(* Schneider Machine Expert - Basic project Motor_StartStop_Overload_TM221CE16T, file version 3.0.0.0 *)
(* ProjectInformations: Name=New project *)

HARDWARE
  Cpu 0: TM221CE16T
  EthernetConfiguration: NetworkName=M221, IpAllocationMode=FixedAddress, IpAddress=0.0.0.0, SubnetMask=0.0.0.0
  SerialLineConfiguration: Baud=Baud19200, Parity=ParityEven, DataBits=DataBits8, StopBits=StopBits1, PhysicalMedium=PhysicalMediumRs485, TransmissionMode=TransmissionModeModbusRtu, SlaveId=1, Addressing=SlaveAddressing
  MastTask: UsePeriodScanMode=false, PeriodScan=100
  FastTask: Period=255
  CpuBehavior: StartingMode=StartAsPreviousState, AutoSaveRamOnEeprom=true, WatchdogPeriod=250

SYMBOLS  (address, symbol, comment, settings)
  %M0       SYSTEM_READY
  %M1       MOTOR_RUNNING
  %M2       OVERLOAD_ALARM
  %M3       ANY_ALARM
  %S0       SB_COLDSTART  "Indicates or executes a cold start (data initialized to default values)"
  %S1       SB_WARMSTART  "Indicates there was a warm start with data backup"
  %TM0        [Preset=3, Base=OneSecond]
  %TM1        [Preset=5, Base=HundredMilliseconds]
  %I0.0     EMERGENCY_PB

POU Motor Control
  (* SectionNumber=0 *)

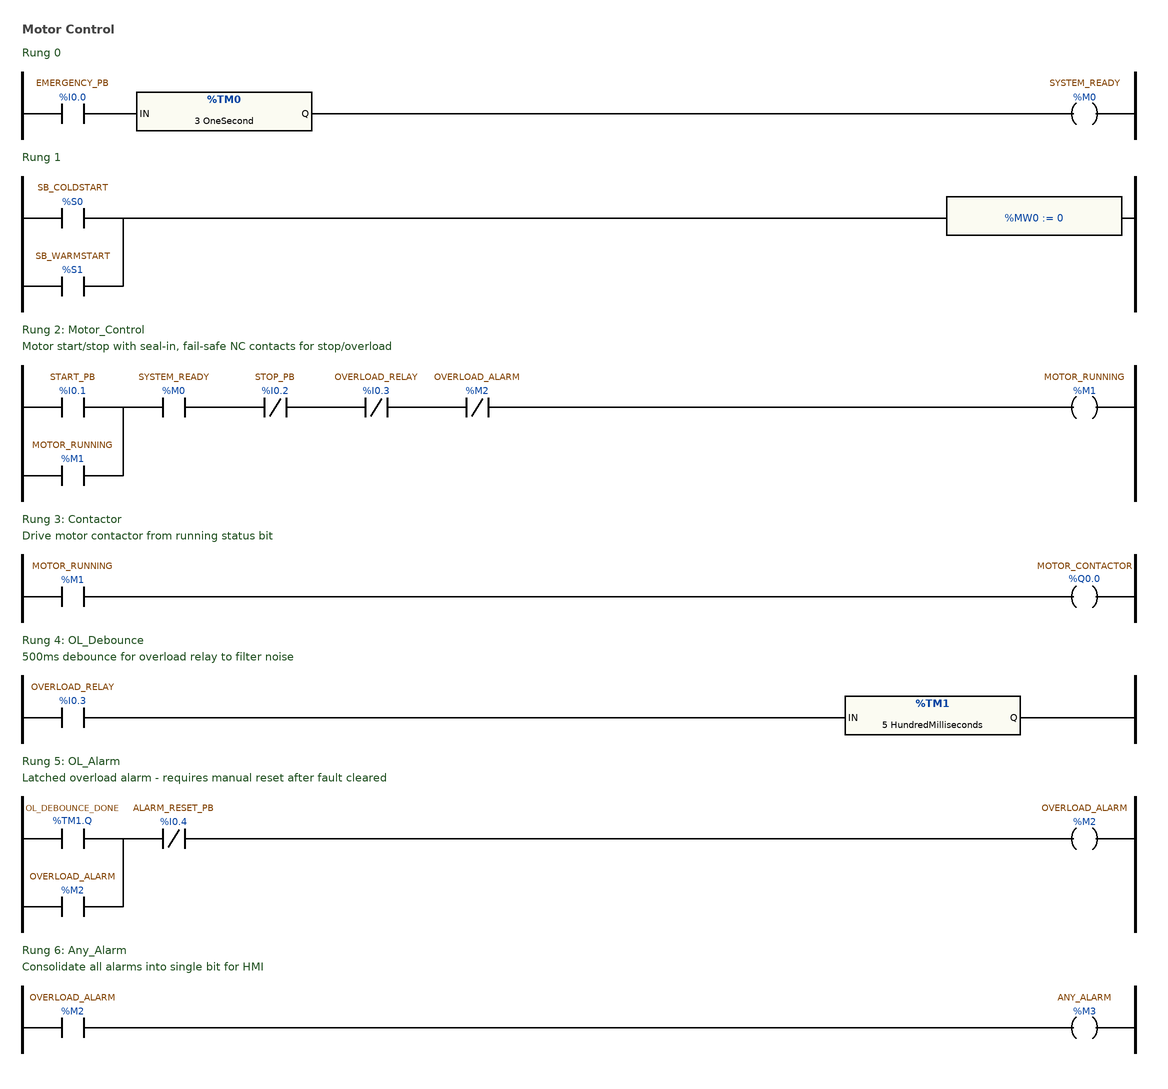

// Rung 0
  BLK %TM0
  LD %I0.0                (* EMERGENCY_PB *)
  IN
  OUT_BLK
  LD Q
  ST %M0                  (* SYSTEM_READY *)
  END_BLK
  // as ST:
  //   %TM0(IN := EMERGENCY_PB);
  //   SYSTEM_READY := %TM0.Q;

// Rung 1
  LD %S0                  (* SB_COLDSTART *)
  OR %S1                  (* SB_WARMSTART *)
  [ %MW0 := 0 ]
  // as ST:
  //   IF SB_COLDSTART OR SB_WARMSTART THEN %MW0 := 0; END_IF;

// Rung 2: Motor_Control
// Motor start/stop with seal-in, fail-safe NC contacts for stop/overload
  LD %I0.1                (* Start Pushbutton *)
  OR %M1                  (* MOTOR_RUNNING - Seal-in *)
  AND %M0                 (* SYSTEM_READY - System Ready *)
  ANDN %I0.2              (* Stop Button NC *)
  ANDN %I0.3              (* Overload OK *)
  ANDN %M2                (* OVERLOAD_ALARM - No Alarm *)
  ST %M1                  (* MOTOR_RUNNING - Motor Running *)
  // %I0.1: Start Pushbutton
  // %M0: System Ready
  // %I0.2: Stop Button NC
  // %I0.3: Overload OK
  // %M2: No Alarm
  // %M1: Motor Running
  // %M1: Seal-in
  // as ST:
  //   MOTOR_RUNNING := (%I0.1 OR MOTOR_RUNNING) AND SYSTEM_READY AND NOT %I0.2 AND NOT %I0.3 AND NOT OVERLOAD_ALARM;

// Rung 3: Contactor
// Drive motor contactor from running status bit
  LD %M1                  (* MOTOR_RUNNING - Motor Running *)
  ST %Q0.0                (* Motor Contactor *)
  // %M1: Motor Running
  // %Q0.0: Motor Contactor
  // as ST:
  //   %Q0.0 := MOTOR_RUNNING;

// Rung 4: OL_Debounce
// 500ms debounce for overload relay to filter noise
  BLK %TM1                (* Overload Debounce Timer *)
  LD %I0.3                (* Overload Relay Tripped *)
  IN
  OUT_BLK
  END_BLK
  // %I0.3: Overload Tripped
  // %TM1: 500ms Debounce
  // as ST:
  //   %TM1(IN := %I0.3);

// Rung 5: OL_Alarm
// Latched overload alarm - requires manual reset after fault cleared
  LD %TM1.Q               (* Debounce Timer Done *)
  OR %M2                  (* OVERLOAD_ALARM - Seal-in Alarm *)
  ANDN %I0.4              (* Reset Not Pressed *)
  ST %M2                  (* OVERLOAD_ALARM - Overload Alarm *)
  // %TM1.Q: Debounce Done
  // %I0.4: Reset Not Pressed
  // %M2: Overload Alarm
  // %M2: Seal-in
  // as ST:
  //   OVERLOAD_ALARM := (%TM1.Q OR OVERLOAD_ALARM) AND NOT %I0.4;

// Rung 6: Any_Alarm
// Consolidate all alarms into single bit for HMI
  LD %M2                  (* OVERLOAD_ALARM - Overload Alarm *)
  ST %M3                  (* ANY_ALARM - Any Alarm *)
  // %M2: Overload Alarm
  // %M3: Any Alarm
  // as ST:
  //   ANY_ALARM := OVERLOAD_ALARM;

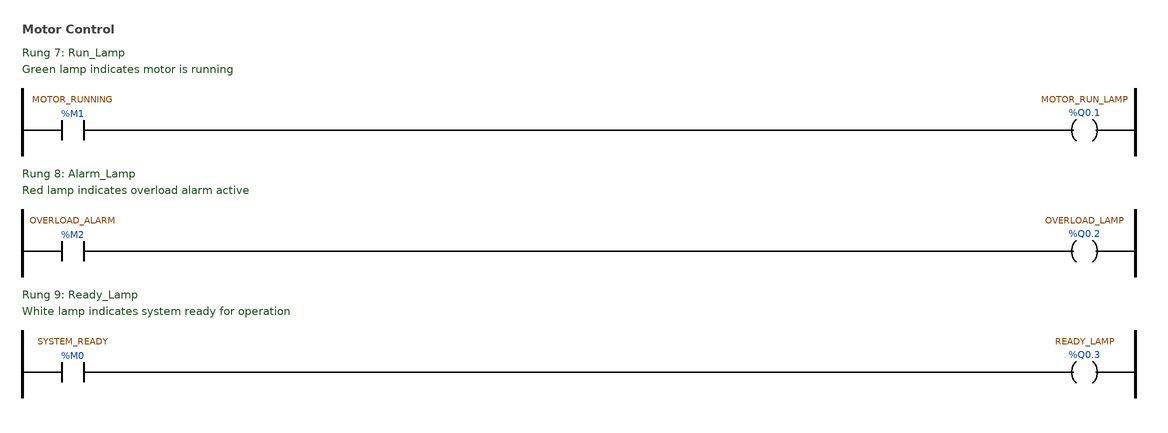

// Rung 7: Run_Lamp
// Green lamp indicates motor is running
  LD %M1                  (* MOTOR_RUNNING - Motor Running *)
  ST %Q0.1                (* Run Lamp *)
  // %M1: Motor Running
  // %Q0.1: Run Lamp
  // as ST:
  //   %Q0.1 := MOTOR_RUNNING;

// Rung 8: Alarm_Lamp
// Red lamp indicates overload alarm active
  LD %M2                  (* OVERLOAD_ALARM - Overload Alarm *)
  ST %Q0.2                (* Alarm Lamp *)
  // %M2: Overload Alarm
  // %Q0.2: Alarm Lamp
  // as ST:
  //   %Q0.2 := OVERLOAD_ALARM;

// Rung 9: Ready_Lamp
// White lamp indicates system ready for operation
  LD %M0                  (* SYSTEM_READY - System Ready *)
  ST %Q0.3                (* Ready Lamp *)
  // %M0: System Ready
  // %Q0.3: Ready Lamp
  // as ST:
  //   %Q0.3 := SYSTEM_READY;
